PROGRAM MAIN
VAR
END_VAR


	PRG_SmartHome();

END_PROGRAM

(* stored: Version 1.1.0.1, ProductVersion 3.1.4024.12
   POU MAIN: Id {7a168334-2e42-47f0-b9cd-ce929aa571b3}, SpecialFunc None *)
